(*
:Description: Writes the given message at the specific level. 

This function implicit uses the global logger ``Const.sGlobalLogger`` with
the value ``'_GLOBAL_'``.

**Example**

.. code:: 

    F_Log(E_LogLevel.eWarn, 'Something important happened.');
	
*)
FUNCTION F_Log
VAR_INPUT
	eLogLevel		: E_LogLevel;		(* The level of this log. *)
	sMessage		: T_MaxString;		(* The message to log. *)
END_VAR
VAR 
	aEmptyArg		: BYTE;
END_VAR

F_LogL(eLogLevel, Const.sGlobalLogger, sMessage);

END_FUNCTION

(* stored: Version 1.1.0.1, ProductVersion 3.1.4024.0
   POU F_Log: Id {000f3ef1-efd9-4a4d-9a1f-6ebbe7a6fe8d}, SpecialFunc None *)
